RoboDK station: Drawing.rdk

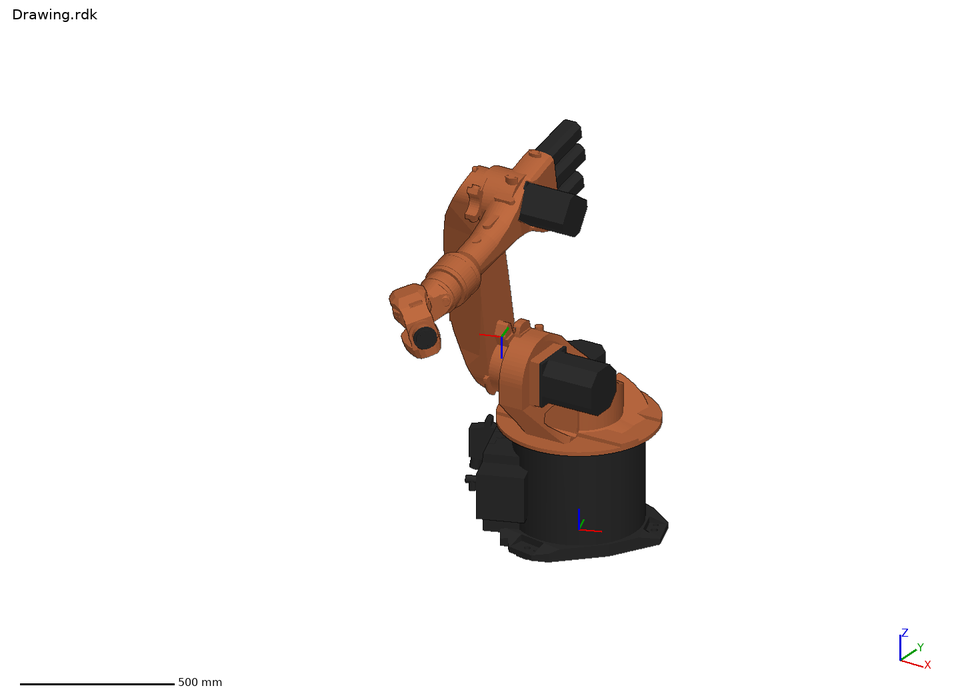
[picture v0: the station drawn from its stored meshes, robots at their saved joint values, targets as dots, program paths as lines]
Station Haploid - Drawing. Poses are relative to the parent item; angles as X-Y-Z fixed-axis rotations.
  - frame KUKA KR 16 2 Base at (-517.2, 80.87, 0) mm, rotated rx 0 ry 0 rz 22.9 deg
    - robot KUKA KR 16 2: 6 axes, payload 16 kg, reach 901 mm, repeatability 0.05 mm, weight 235 kg
        modified DH rows (alpha deg, a mm, theta deg, d mm): 0, 0, 0, 675; -90, 260, 0, 0; 0, 680, -90, 0; -90, -35, 0, 670; 90, 0, 0, 0; -90, 0, 180, 158
        joint limits [-185, -155, -130, -350, -130, -350] to [185, 35, 154, 350, 130, 350]; home [0, -90, 90, 0, 0, 0]; saved at [108.919, -79.886, 90.126, 258.117, 45.075, 5.684]
      - tool Tool, TCP at (0, 0, 100) mm, rotated rx -90 ry 30 rz 170 deg
  - frame Frame draw at (-170.73, -850.83, 1162.99) mm, rotated rx -179.07 ry 0.45 rz -162.16 deg
